(* CODESYS project Untitled1.project

Project tree, tasks and I/O mapping:
  Device : CODESYS Control Win V3, 3S - Smart Software Solutions GmbH, order no. 305021, version 3.5.11.30
    application Application
      libraries: Standard, * (System)
      task MainTask (cyclic, interval t#20ms, priority 1) calls PLC_PRG
      program PLC_PRG [LD]
*)

// Device/Application/PLC_PRG
PROGRAM PLC_PRG
VAR
	B1 : BOOL;      // AVACO DA ESTEIRA
	K1 : BOOL;      // MOTOR DA ESTEIRA
	S3 : BOOL;      // SENSOR DO FIM DA ESTEIRA
	S1: BOOL;       // SENSOR DO INICIO DA ESTEIRA
	S2: BOOL;       // SENSOR DO MEIO DA ESTEIRA
	B2 : BOOL;      // PARA A ESTEIRA
	K2: BOOL;       // INVERSAO DO MOTOR
END_VAR

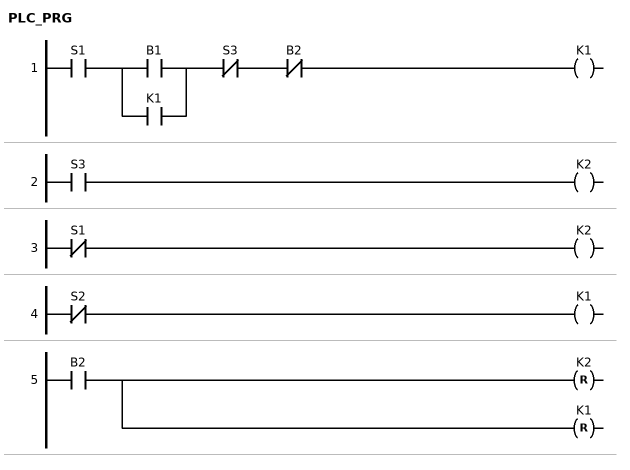
// NETWORK 1
K1 := S1 AND (B1 OR K1) AND NOT S3 AND NOT B2;

// NETWORK 2
K2 := S3;

// NETWORK 3
K2 := NOT S1;

// NETWORK 4
K1 := NOT S2;

// NETWORK 5
K2 R= B2;
K1 R= B2;

END_PROGRAM
